{attribute 'GeneratedUsingTerminal: AX8108-0100-0101-0101'}
{attribute addProperty BoxType "AX8108-0100-0101-0101"}
{attribute addProperty Id "FSOEAT %I*FSOE_3C294B218"}
{attribute addProperty CRC "4258349930"}
{attribute addProperty Size "8"}
TYPE Standard_Inputdata_FDD1436A :
STRUCT
	{attribute addProperty Name "FSOE"}
	FSOE AT %I* : FSOE_3C294B21;
END_STRUCT
END_TYPE

(* stored: Version 1.2.0.0, ProductVersion 3.1.4024.9
   DUT Standard_Inputdata_FDD1436A: Id {f14c4695-8673-4eb7-ac37-eea664eda8d3} *)
